INTERFACE I_MetadatumAddedEvent EXTENDS I_Event

PROPERTY PUBLIC TargetMetadatum : I_Metadatum
GET
END_GET
END_PROPERTY

END_INTERFACE

(* stored: Version 1.1.0.1, ProductVersion 3.1.4024.12
   Itf I_MetadatumAddedEvent: Id {14da0805-61d3-0e9e-3d26-198dbf34f884}
   Property TargetMetadatum: Id {cd61a1c6-2dea-0766-3eef-884b65dc73f2}
   Get Get: Id {b0d09e0c-a50d-021c-26ea-e911450dd15c} *)
